(* IEC 61131-3 sources: CodesysTest/export/UN00 - Sharp Bagger/EM01 - Bagger Head/CM07 - IBD/FB_BaseIBD.pou, 2 files *)

(* ---- FB_BaseIBD.pou.st ---- *)
(*#-#-#-#-#-#-#-#-#-#---Declaration---#-#-#-#-#-#-#-#-#-#-#-#-#*)

FUNCTION_BLOCK FB_BaseIBD EXTENDS FB_BaseComponent IMPLEMENTS I_IBD
VAR_INPUT
END_VAR
VAR_OUTPUT
END_VAR
VAR
	_MoveInToDeflate : BOOL;
	_MoveOut : BOOL;
	_RemovePower : BOOL;
END_VAR
(*#-#-#-#-#-#-#-#-#-#---Implementation---#-#-#-#-#-#-#-#-#-#-#-#-#*)

SUPER^();

(* ---- RemovePower.m.st ---- *)
(*#-#-#-#-#-#-#-#-#-#---Declaration---#-#-#-#-#-#-#-#-#-#-#-#-#*)

METHOD RemovePower
VAR_INPUT
END_VAR
(*#-#-#-#-#-#-#-#-#-#---Implementation---#-#-#-#-#-#-#-#-#-#-#-#-#*)

_RemovePower := TRUE;
